{attribute 'no_explicit_call' := 'do not call this POU directly, call execute'} 
FUNCTION_BLOCK _TemplateFB_1
VAR
END_VAR

// NO CODE HERE, USE execute

METHOD execute
END_METHOD

END_FUNCTION_BLOCK

(* stored: Version 1.1.0.1
   POU _TemplateFB_1: Id {02158913-a73f-4837-9272-0eaa1d312448}, SpecialFunc None
   Method execute: Id {b8daca9b-cfc4-4f3a-99b0-54786a5f28e0} *)
